// TIA Portal V16 export
// export: Created 2022-02-28T20:47:28.7287533Z, ExportSetting WithDefaults, DisplayName Totally Integrated Automation Portal, DisplayVersion V16, DisplayName TIA Portal Version Control Interface, DisplayVersion V16, DisplayName TIA Portal Openness, DisplayVersion V16, DisplayName STEP 7 Professional, DisplayVersion V16, DisplayName STEP 7 Safety, DisplayVersion V16, DisplayName WinCC Advanced, DisplayVersion V16
VAR_GLOBAL   // PLC tag table "02_Camara_1"
   "DataMan-TriggerEnable" AT %Q200.0 : Bool;
   "DataMan-Trigger" AT %Q200.1 : Bool;
   "DataMan-TriggerReady" AT %I200.0 : Bool;
   "DataMan-TriggerAck" AT %I200.1 : Bool;
   "DataMan-Acquiring" AT %I200.2 : Bool;
   "DataMan-MissedAcq" AT %I200.3 : Bool;
   "DataMan-TriggerID" AT %IW201 : Word;
   "DataMan-BufferResultsEnable" AT %Q300.0 : Bool;
   "DataMan-ResultsAck" AT %Q300.1 : Bool;
   "DataMan-Decoding" AT %I500.0 : Bool;
   "DataMan-Decode Complete" AT %I500.1 : Bool;
   "DataMan-Results Buffer Overrun" AT %I500.2 : Bool;
   "DataMan-Results Available" AT %I500.3 : Bool;
   "DataMan-General Fault" AT %I500.7 : Bool;
   "DataMan-Train Code" AT %Q600.0 : Bool;
   "DataMan-Train Match String" AT %Q600.1 : Bool;
   "DataMan-Train Focus" AT %Q600.2 : Bool;
   "DataMan-Train Brightness" AT %Q600.3 : Bool;
   "DataMan-Untrain" AT %Q600.4 : Bool;
   "DataMan-Execute DMCC" AT %Q600.6 : Bool;
   "DataMan-Set Match String" AT %Q600.7 : Bool;
   "DataMan-Train Code Ack" AT %I400.0 : Bool;
   "DataMan-Train Match String Ack" AT %I400.1 : Bool;
   "DataMan-Train Focus Ack" AT %I400.2 : Bool;
   "DataMan-Train Brightness Ack" AT %I400.3 : Bool;
   "DataMan-Untrain Ack" AT %I400.4 : Bool;
   "DataMan-Execute DMCC Ack" AT %I400.6 : Bool;
   "DataMan-Set Match String Ack" AT %I400.7 : Bool;
   "DataMan-UserData Option" AT %QW500 : Word;
   "DataMan-UserData Length" AT %QW502 : Word;
   "DataMan-UserData[0]" AT %QB504 : Byte;
   "DataMan-UserData[1]" AT %QB505 : Byte;
   "DataMan-UserData[2]" AT %QB506 : Byte;
   "DataMan-UserData[3]" AT %QB507 : Byte;
   "DataMan-UserData[4]" AT %QB508 : Byte;
   "DataMan-UserData[5]" AT %QB509 : Byte;
   "DataMan-UserData[6]" AT %QB510 : Byte;
   "DataMan-UserData[7]" AT %QB511 : Byte;
   "DataMan-UserData[8]" AT %QB512 : Byte;
   "DataMan-UserData[9]" AT %QB513 : Byte;
   "DataMan-UserData[10]" AT %QB514 : Byte;
   "DataMan-UserData[11]" AT %QB515 : Byte;
   "DataMan-UserData[12]" AT %QB516 : Byte;
   "DataMan-UserData[13]" AT %QB517 : Byte;
   "DataMan-UserData[14]" AT %QB518 : Byte;
   "DataMan-UserData[15]" AT %QB519 : Byte;
   "DataMan-ResultID" AT %IW700 : Word;
   "DataMan-Result Code" AT %IW702 : Word;
   "DataMan-Result Extended" AT %IW704 : Word;
   "DataMan-Result Length" AT %IW706 : Word;
   "DataMan-InspectionResults[0]" AT %IB708 : Byte;
   "DataMan-InspectionResults[1]" AT %IB709 : Byte;
   "DataMan-InspectionResults[2]" AT %IB710 : Byte;
   "DataMan-InspectionResults[3]" AT %IB711 : Byte;
   "DataMan-InspectionResults[4]" AT %IB712 : Byte;
   "DataMan-InspectionResults[5]" AT %IB713 : Byte;
   "DataMan-InspectionResults[6]" AT %IB714 : Byte;
   "DataMan-InspectionResults[7]" AT %IB715 : Byte;
   "DataMan-InspectionResults[8]" AT %IB716 : Byte;
   "DataMan-InspectionResults[9]" AT %IB717 : Byte;
   "DataMan-InspectionResults[10]" AT %IB718 : Byte;
   "DataMan-InspectionResults[11]" AT %IB719 : Byte;
   "DataMan-InspectionResults[12]" AT %IB720 : Byte;
   "DataMan-InspectionResults[13]" AT %IB721 : Byte;
   "DataMan-InspectionResults[14]" AT %IB722 : Byte;
   "DataMan-InspectionResults[15]" AT %IB723 : Byte;
END_VAR
